(* IEC 61131-3 sources: 1326_JeddahAppartment/1326 - Jeddah Appartment - Last/PLC3_Somfy, 3 files *)

(* ---- PLC3_SOMFY.ST ---- *)
TYPE
  TCurtainStatus : Struct
    outUP   : BOOl;
    outDW   : BOOl;
    pos     : USINT;
    normPos : USINT;
  End_Struct;
END_TYPE

TYPE
   TEnCurtain : Struct
      UP   : BOOL;
      DW   : BOOl;
      STOP : BOOL;
   End_Struct;
END_TYPE

VAR_GLOBAL CONSTANT
   numOfCurtains      : USINT := 14;
   numOfCurtains_PLC1 : USINT := 9;
   numOfCurtains_PLC2 : USINT := 5;
   curtUpDwTime      : TIME := T#18s;
END_VAR

VAR_GLOBAL
  curtainsStatus AT PLC3.DATA : Array[1..numOfCurtains] of TCurtainStatus;
  PLC1_EnCurtains AT PLC1_Curtains.DATA : Array[1..numOfCurtains_PLC1] of TEnCurtain;
  PLC2_EnCurtains AT PLC2_Curtains.DATA : Array[1..numOfCurtains_PLC2] of TEnCurtain;
END_VAR

(* ---- fbSomfyRTSControl.ST ---- *)
VAR_GLOBAL CONSTANT
   BUFFER_SIZE : UINT := 5;
END_VAR

TYPE
   TSomfyRTSPacket : Struct
         packet : Array[0..15] of USINT;
         length : UINT;
   End_Struct;

   TSomfyRTSPacketBuff : Array[1..BUFFER_SIZE] of TSomfyRTSPacket;

   TVendorID       : Array[1..3] of USINT;
   TSomfyCtrl      : struct
        UP, DW, favPos, stop , setChannel : Bool;
        openProg : BOOL;
        set_IP : BOOL;
   End_struct;
END_TYPE

//==========================================================================

FUNCTION somfyBuffer_Push : BOOL
  VAR_INPUT
  newPacket  : TSomfyRTSPacket;
  END_VAR

  VAR_IN_OUT
  buffer : TSomfyRTSPacketBuff;
  index  : UINT;
  END_VAR
  VAR

  END_VAR

  VAR_TEMP
  emptyPacket : TSomfyRTSPacket;
  END_VAR

  if index < BUFFER_SIZE then
     if newPacket <> emptyPacket then
       index := index + 1;
       buffer[index] := newPacket;
       somfyBuffer_Push := 1;
     else
       somfyBuffer_Push := 0;
     end_if;
  else
     somfyBuffer_Push := 0;
  end_if;

END_FUNCTION

//===========================================================================

FUNCTION somfyBuffer_Pop : TSomfyRTSPacket
  VAR_IN_OUT
  buffer : TSomfyRTSPacketBuff;
  index  : UINT;
  END_VAR

  VAR_TEMP
  i : UINT;
  popedPacket : TSomfyRTSPacket;
  END_VAR

  if index > 0 then
     popedPacket := buffer[1];
     for i := 1 to BUFFER_SIZE-1 do
         buffer[i] :=  buffer[i+1];
     end_for;
     index := index - 1;
  end_if;
  somfyBuffer_Pop := popedPacket;

END_FUNCTION

//===========================================================================

FUNCTION fbSomfyRTS_Cmnd : BOOL
  // Push new RTS control packet to the buffer according to the action input
  // the buffer should be passed to fbSomfyRTSCtrl function block to execute its commands
  VAR_INPUT
  ChNum         : USINT;
  HostID        : TVendorID;    // 3 hex bytes address set for PLC as non Somfy host
  TrsnsmitterID : TVendorID;    // ID of Transmitter written on the product

  UP, DW, favPos, stop , setChannel : Bool;
  openProg : BOOL;
  set_IP : BOOL;
  END_VAR

  VAR_IN_OUT
  //somfyCtrl     : TSomfyCtrl;
  packetsBuffer :  TSomfyRTSPacketBuff;
  buffIndex     : UINT;
  END_VAR

  VAR
  packet      : TSomfyRTSPacket;
  END_VAR

  VAR_TEMP
  length      : UINT := 2;
  i           : usint;
  frameChksum : USINT;
  END_VAR

  packet.packet[2] := 16#FA;

  if UP or DW or favPos or stop then
     packet.packet[0] := 16#7f;
     packet.packet[1] := 16#72;
     packet.packet[11] := 16#06;
     length := 13;
  elsif setChannel then
     packet.packet[0] := 16#68;
     packet.packet[1] := 16#73;
     packet.packet[10] := 16#05;
     length := 12;
     //setChannel := 0;
  elsif openProg then
     packet.packet[0] := 16#67;
     packet.packet[1] := 16#73;
     packet.packet[10] := 16#05;
     length := 12;
     //openProg := 0;
  elsif set_IP then
     packet.packet[0] := 16#65;
     packet.packet[1] := 16#73;
     packet.packet[10] := 16#05;
     length := 12;
     //set_IP := 0;
  end_if;

  if UP then
     packet.packet[10] := 16#FE;
     //UP := 0;
  elsif DW then
     packet.packet[10] := 16#FD;
     //DW := 0;
  elsif stop then
     packet.packet[10] := 16#FC;
  elsif favPos then
     packet.packet[10] := 16#FB;
     //favPos := 0;
  end_if;

  packet.packet[9] :=  255 -  ChNum;

  for i := 3 to 5  do
      packet.packet[i] := 255 - HostID[i-2];
  end_for;
  for i := 6 to 8  do
      packet.packet[i] := 255 - TrsnsmitterID[i-5];
  end_for;

  frameChksum := CheckSum(ptr := adr(packet) , length := length-2);
  packet.packet[length-1] := frameChksum;
  packet.length := length;

  if somfyBuffer_Push(newPacket := packet, buffer := packetsBuffer, index := buffIndex) then
     fbSomfyRTS_Cmnd := 0;
  else
     fbSomfyRTS_Cmnd := 1;
  end_if;

END_FUNCTION

//========================================================================================

FUNCTION_BLOCK fbSomfyRTSCtrl
  VAR_INPUT
  En      : BOOL;
  CH_ID   : UINT;
  END_VAR

  VAR_OUTPUT
  Err : USINT;
  ErrText : String;
  END_VAR

  VAR_IN_OUT
  packetsBuffer :  TSomfyRTSPacketBuff;
  buffIndex     : UINT;
  END_VAR

  VAR
  packet      : TSomfyRTSPacket;
  RQ          : BOOL;

  sendTimer   : fbTick;
  send        : fbSendTo;

  END_VAR

  VAR_TEMP
  emptyPacket : TSomfyRTSPacket;
  END_VAR

  sendTimer(IN := En and (buffIndex > 0) , PT := T#500ms);

  if sendTimer.Q then
     packet := somfyBuffer_Pop(buffer := packetsBuffer, index := buffIndex);
     if packet <> emptyPacket then
        RQ := 1;
     end_if;
  end_if;

  send(rq := En and RQ, chanCode := CH_ID, lenTx := packet.length, data := void(packet.packet), error => Err);
  if send.mesSent or Err > 0 then
     RQ := 0;
  end_if;

  if En then
      Err := send.error;
  else
      Err := 0;
  end_if;

  ErrText := GetLastComErrTxt(errCode := Err);

END_FUNCTION_BLOCK

(* ---- prgMain.ST ---- *)
VAR_GLOBAL RETAIN
   curtainsFB    : Array[1..numOfCurtains] of fb_iJalousie;
   packetsBuffer : TSomfyRTSPacketBuff;
   buffIndex     : UINT;
END_VAR

TYPE
   TEnCurtainRT : Struct
     UP   : R_TRIG;
     DW   : R_TRIG;
     STOP : R_TRIG;
   End_Struct;
END_TYPE

PROGRAM prgMain
  VAR_INPUT
  END_VAR
  VAR_OUTPUT
  END_VAR
  VAR
  EnCurtains    : Array[1..numOfCurtains] of TEnCurtain;
  EnCurtains_RT : Array[1..numOfCurtains] of TEnCurtainRT;

  i : USINT;
  curIndex : USINT;

  Trsnsmitter1_ID ,Trsnsmitter2_ID : TVendorID;
  HostID : TVendorID;

  somfyRTSCtrl_Master : fbSomfyRTSCtrl;

  // for test
  test, up, dw, stop, block : BOOl;
  up_RT , dw_RT : R_TRIG;

  END_VAR
  VAR_TEMP
  END_VAR

  for i := 1 to numOfCurtains do
      if i <= numOfCurtains_PLC1 then
         EnCurtains[i] := PLC1_EnCurtains[i];
      else
         EnCurtains[i] := PLC2_EnCurtains[i - numOfCurtains_PLC1];
      end_if;

      EnCurtains_RT[i].UP(CLK := EnCurtains[i].UP);
      EnCurtains_RT[i].DW(CLK := EnCurtains[i].DW);
      EnCurtains_RT[i].STOP(CLK := EnCurtains[i].STOP);

      // Generate RTS control packets
      if EnCurtains_RT[i].UP.Q then
         fbSomfyRTS_Cmnd(ChNum := i, HostID := HostID, TrsnsmitterID := Trsnsmitter1_ID, UP := 1,  packetsBuffer := packetsBuffer, buffIndex := buffIndex);
      end_if;

       if EnCurtains_RT[i].DW.Q then
         fbSomfyRTS_Cmnd(ChNum := i, HostID := HostID, TrsnsmitterID := Trsnsmitter1_ID, DW := 1,  packetsBuffer := packetsBuffer, buffIndex := buffIndex);
      end_if;

       if EnCurtains_RT[i].STOP.Q then
         fbSomfyRTS_Cmnd(ChNum := i, HostID := HostID, TrsnsmitterID := Trsnsmitter1_ID, stop := 1,  packetsBuffer := packetsBuffer, buffIndex := buffIndex);
      end_if;

      // handle curtains status
      if (EnCurtains_RT[i].UP.Q and curtainsFB[i].outDw) or (EnCurtains_RT[i].DW.Q and curtainsFB[i].outUp) then
         curtainsFB[i].up := 0;
         curtainsFB[i].dw := 0;
         curtainsFB[i](stop := 1, upDwTime := curtUpDwTime) ;
      else
         curtainsFB[i](up := EnCurtains[i].UP, dw := EnCurtains[i].DW, stop := EnCurtains[i].STOP, upDwTime := curtUpDwTime) ;
      end_if;

      curtainsStatus[i].outUP   := curtainsFB[i].outUp;
      curtainsStatus[i].outDW   := curtainsFB[i].outDw;
      curtainsStatus[i].pos     := 100 - curtainsFB[i].posit;
      curtainsStatus[i].normPos := curtainsStatus[i].pos / 25;

  end_for;

  somfyRTSCtrl_Master(En := true, CH_ID := CH2_UNI, packetsBuffer := packetsBuffer, buffIndex := buffIndex);

 (*
  up_RT(CLK := up);
  dw_RT(CLK := dw);

  if (up_RT.Q and curtainsFB[1].outDw) or (dw_RT.Q and curtainsFB[1].outUp) then
     curtainsFB[1].up := 0;
     curtainsFB[1].dw := 0;
     curtainsFB[1](stop := 1, upDwTime := curtUpDwTime) ;
     test := 1;
  else
     curtainsFB[1](up := up, dw := dw, stop := STOP, upDwTime := curtUpDwTime) ;
     up   := 0;
     dw   := 0;
     stop := 0;
  end_if;  *)

END_PROGRAM
